TYPE T_CodePIT : STRING[7];
END_TYPE

(* stored: Version 1.1.0.1
   DUT T_CodePIT: Id {47d48b82-5bf8-4169-a77e-1d9687ddea1b} *)
